FUNCTION_BLOCK HYST_2
VAR_INPUT
	IN : REAL;
	VAL : REAL;
	HYS : REAL;
END_VAR
VAR_OUTPUT
	Q : BOOL;
	WIN: BOOL;
END_VAR
VAR
	tmp: REAL;
END_VAR


(*
version 1.2	2. jun. 2008
programmer 	oscat
tested BY	oscat

this hysteresis function switches the output high if the input signal reaches obove val + hys/2 and will switch to low when the input falls back below val - hys/2 value.
a separate output mid is set if the input stays between low and high value.

*)

tmp := val - hys * 0.5;
IF in < tmp THEN
	Q := FALSE;
	win := FALSE;
ELSIF in > tmp + hys THEN
	Q := TRUE;
	win := FALSE;
ELSE
	win := TRUE;
END_IF;



(* revision history
hm		4. aug 2006	rev 1.0
	original version

hm		5. jan 2008	rev 1.1
	improved code for better performance

hm		2. jun. 2008	rev 1.2
	improved performance
*)

END_FUNCTION_BLOCK

(* stored: Version 1.1.0.1, ProductVersion 3.1.4024.9
   POU HYST_2: Id {34905041-e76b-448f-a1a8-841016f26873}, SpecialFunc None *)
